(* IEC 61131-3 sources: s22-soft-shell/st_interpret/tests/test_inputs/st_subset_1, 12 files *)

(* ---- 01_Bool.st ---- *)
PROGRAM 01_real
    VAR
		a : bool;
    END_VAR
		a := TRUE;
END_PROGRAM

(* ---- 01_Bool_01.st ---- *)
PROGRAM 01_real //boolean accepts integers 0 and 1
    VAR
	a : bool;
        b : bool;
        c : bool;
        d : bool;
    END_VAR
	a := TRUE;
        b := FALSE;
        c := 1; //true
        d := 0; //false

END_PROGRAM

(* ---- 01_Int.st ---- *)
PROGRAM 01_Int
    VAR
		a : INT;
    END_VAR
		a := 1;
END_PROGRAM

(* ---- 01_mixed.st ---- *)
PROGRAM 01_real //accepts all types in same program
    VAR
	a : real;
        b : int;
        c : bool;
    END_VAR
	a := 1.2;
        b := 5;
        c := True;
END_PROGRAM

(* ---- 01_Multi.st ---- *)
PROGRAM 01_Multi
    VAR
        a : INT;
        b : INT;
        c : INT;
    END_VAR
        a := 1;
        b := 2;
        c := 3;
END_PROGRAM

(* ---- 01_NestedBool.st ---- *)
PROGRAM 01_NestedBool
    VAR
	a : bool;
        b : bool;
        c : bool;
    END_VAR
	a := true;
        b := a;
        c := b;
END_PROGRAM

(* ---- 01_NestedInt.st ---- *)
PROGRAM 01_NestedInt
    VAR
	a : INT;
        b : INT;
        c : INT;
    END_VAR
 	a := 1;
        b := a;
        c := b;
END_PROGRAM

(* ---- 01_NestedReal.st ---- *)
PROGRAM 01_NestedReal
    VAR
	a : real;
        b : real;
        c : real;
    END_VAR
	a := 1.5;
        b := a;
        c := b;
END_PROGRAM

(* ---- 01_Real.st ---- *)
PROGRAM 01_real
    VAR
		a : real;
    END_VAR
		a := 1.2;
END_PROGRAM

(* ---- 01_truncate.st ---- *)
PROGRAM 01_truncate //should not error but rather truncate 1.5 to 1
    VAR
	a : INT;
    END_VAR
	a := 1.5;
END_PROGRAM

(* ---- BlockComments.st ---- *)
(* block comment *) (* multiline
block comment *)
PROGRAM blockComments(* block comment *) (* multiline
block comment *)
    VAR (* block comment *) (* multiline
block comment *)
		a : INT;(* block comment *) (* multiline
block comment *)
    END_VAR(* block comment *) (* multiline
block comment *)
		a (* block comment *) :=  (* block comment *) 1;(* block comment *) (* multiline
block comment *)
    b := 5;(* block comment *) (* multiline
block comment *)
END_PROGRAM(* block comment *) (* multiline
block comment *)
(* block comment *) (* multiline
block comment *)

(* ---- LineComments.st ---- *)
// line comment
PROGRAM lineComments // line comment
    // line comment
    VAR  // line comment
		a : INT;  // line comment
    // line comment
    b : INT;  // line comment
    // line comment
    END_VAR // line comment
    // line comment
		a := 1;  // line comment
    // line comment
    b := 5; // line comment
    // line comment
END_PROGRAM // line comment
// line comment
